# EPICS substitutions: IOCs/12id/iocBoot/ioc12ida2/standardScans.substitutions
file "$(SSCAN)/sscanApp/Db/standardScans.db"
{
pattern
{P, MAXPTS1, MAXPTS2, MAXPTS3, MAXPTS4, MAXPTSH}
{12ida2:, 8000, 1000, 1000, 1000, 8000}
}
